FUNCTION_BLOCK T_RoboConnect_Enable_RobotEnabled EXTENDS T_UnitTestBase
VAR
  _robot : I_RoboConnect;
  myTestState, prevState : (ARRANGE, ACT, ASSERT);
  actual : STRING;
  expected : STRING := '0';
  resultTask : I_Task;
END_VAR

CASE myTestState OF
  ARRANGE:
    StateChanged();
    myTestState := ACT;

  ACT:
  IF StateChanged() THEN
    _robot.Enable(task => resultTask);
    
	ELSIF NOT resultTask.Busy THEN
        myTestState := ASSERT;
  END_IF
  
  ASSERT:
    actual := resultTask.ErrorId;
    assertion.AssertEquals_STRING(expected, actual, 'actual := _robot.Enabled;');
    myTestState := ARRANGE;
    TestFinished();
END_CASE

METHOD FB_init : BOOL
VAR_INPUT
  bInitRetains : BOOL; // if TRUE, the retain variables are initialized (warm start / cold start)
  bInCopyCode : BOOL; // if TRUE, the instance afterwards gets moved into the copy code (online change)
  TestSuite : I_TestSuite;
  robot : I_TcRobot;
END_VAR
_robot := robot;
END_METHOD

METHOD PRIVATE StateChanged : BOOL
IF  myTestState = prevState THEN
  RETURN;
END_IF

prevState := myTestState;
StateChanged := TRUE;
END_METHOD

METHOD WaitForCycles : BOOL
VAR_INPUT
  maxCount : UINT;
END_VAR
counter := counter + 1;

IF counter = maxCount THEN
  counter := 0;
  WaitForCycles := TRUE;
END_IF
END_METHOD

END_FUNCTION_BLOCK

(* stored: Version 1.1.0.1
   POU T_RoboConnect_Enable_RobotEnabled: Id {9a50edd7-1b34-4c32-aa9b-2a7aa64e8fc3}, SpecialFunc None
   Method FB_init: Id {65e75648-f731-4da3-846d-dc8f195aa771}
   Method StateChanged: Id {a774d502-a52d-4074-9b02-c30dc15147f6}
   Method WaitForCycles: Id {b5a4e1e1-cf33-4121-a3bf-2d114269b329} *)
